# EPICS autosave request: support/ip/2-9/ipApp/Db/Eurotherm2k_settings.req
$(P)$(TC):RBV_pvTemp.DESC
$(P)$(TC):Setpoint.VAL
$(P)$(TC):RampRate.VAL
$(P)$(TC):P
$(P)$(TC):I
$(P)$(TC):D
